(* IEC 61131-3 sources: repolevel_ST_code_completion/ground_truth/repoeval_can/readful_result, 4 files *)

(* ---- CAN_Send_Data_SWMC.st ---- *)
It seems like you've pasted a portion of the code multiple times, and it is incomplete in some places. However, I can help you analyze and understand the structure of the `CAN_Send_Data_SWMC` function based on the provided fragments.

### Overview of the `CAN_Send_Data_SWMC` Function

The `CAN_Send_Data_SWMC` function is designed to send CAN (Controller Area Network) messages based on the `SWMC_ID` input. It uses a `CASE` statement to determine which CAN channel (`C1`, `C2`, `C3`, etc.) to use for transmitting the message. The function takes the following inputs:
- `SWMC_ID`: A `UINT` value that determines which CAN channel to use.
- `id`: A `UINT` value used to calculate the `TxMsg_CobId`.
- `data`: An array of 8 bytes representing the data to be transmitted.

### Key Observations
1. **Message Structure**:
   - Each CAN channel (e.g., `C1TxMsg`, `C2TxMsg`, etc.) has a `TxMsg_CobId` and `TxMsg_Byte` field.
   - The `TxMsg_CobId` is calculated as `8 + 32 * id`.
   - The `TxMsg_Byte` is assigned the `data` array.

2. **Message Count and Counter**:
   - The `NoOfTxMessages` is set to `1` for each channel, indicating that one message is being transmitted.
   - The `TxCounter` is incremented by 1 for each transmission, likely to keep track of the number of messages sent.

3. **SWMC_ID Handling**:
   - The `CASE` statement handles different `SWMC_ID` values (e.g., `1`, `2`, `3`, `4`).
   - For each `SWMC_ID`, the corresponding CAN channel is selected, and the message is prepared for transmission.

### Issues in the Provided Code
1. **Incomplete Code**:
   - The code fragments are incomplete, with some parts cut off (e.g., the last fragment ends abruptly with `gCan.C1`).

2. **Redundancy**:
   - The same logic is repeated for each `SWMC_ID`. This could be refactored to reduce redundancy and improve maintainability.

3. **Missing Return Value**:
   - The function is declared to return a `BOOL`, but the return value is not shown in the provided code. It is unclear what the function should return (e.g., success/failure of the transmission).

### Refactored Version
Here’s a refactored version of the function to reduce redundancy:

```st
FUNCTION CAN_Send_Data_SWMC : BOOL
VAR_INPUT
	SWMC_ID : UINT;
	id 		: UINT;
	data	: ARRAY[1..8] OF BYTE;
END_VAR
VAR
	txMsgPointer : POINTER TO gCan.C1TxMsg; // Generic pointer to CAN message structure
END_VAR

CASE SWMC_ID OF
	1: txMsgPointer := ADR(gCan.C1TxMsg);
	2: txMsgPointer := ADR(gCan.C2TxMsg);
	3: txMsgPointer := ADR(gCan.C3TxMsg);
	4: txMsgPointer := ADR(gCan.C4TxMsg);
	ELSE
		RETURN FALSE; // Invalid SWMC_ID
END_CASE;

// Set message parameters
txMsgPointer^.TXMsg[1].TxMsg_CobId := 8 + 32 * id;
txMsgPointer^.TXMsg[1].TxMsg_Byte := data;
txMsgPointer^.NoOfTxMessages := 1;
txMsgPointer^.TxCounter := txMsgPointer^.TxCounter + 1;

RETURN TRUE; // Transmission setup successful
```

### Explanation of Refactored Code
1. **Generic Pointer**:
   - A pointer (`txMsgPointer`) is used to reference the appropriate CAN message structure (`C1TxMsg`, `C2TxMsg`, etc.) based on `SWMC_ID`.

2. **Error Handling**:
   - If an invalid `SWMC_ID` is provided, the function returns `FALSE`.

3. **Reduced Redundancy**:
   - The message preparation logic is written only once, reducing code duplication.

4. **Return Value**:
   - The function returns `TRUE` if the message setup is successful, or `FALSE` if an invalid `SWMC_ID` is provided.

Let me know if you need further clarification or assistance!

(* ---- CAN_Send_Data_SWMC_1.st ---- *)
It seems like you've pasted a portion of the code multiple times, and it is incomplete in some places. However, I can help you analyze and understand the structure of the `CAN_Send_Data_SWMC` function based on the provided fragments.

### Overview of the `CAN_Send_Data_SWMC` Function

The `CAN_Send_Data_SWMC` function is designed to send CAN (Controller Area Network) messages based on the `SWMC_ID` input. It uses a `CASE` statement to determine which CAN channel (`C1`, `C2`, `C3`, etc.) to use for transmitting the message. The function takes the following inputs:
- `SWMC_ID`: A `UINT` value that determines which CAN channel to use.
- `id`: A `UINT` value used to calculate the `TxMsg_CobId`.
- `data`: An array of 8 bytes representing the data to be transmitted.

### Key Observations
1. **Message Structure**:
   - Each CAN channel (e.g., `C1TxMsg`, `C2TxMsg`, etc.) has a `TxMsg_CobId` and `TxMsg_Byte` field.
   - The `TxMsg_CobId` is calculated as `8 + 32 * id`.
   - The `TxMsg_Byte` is assigned the `data` array.

2. **Message Count and Counter**:
   - The `NoOfTxMessages` is set to `1` for each channel, indicating that one message is being transmitted.
   - The `TxCounter` is incremented by 1 for each transmission, likely to keep track of the number of messages sent.

3. **SWMC_ID Handling**:
   - The `CASE` statement handles different `SWMC_ID` values (e.g., `1`, `2`, `3`, `4`).
   - For each `SWMC_ID`, the corresponding CAN channel is selected, and the message is prepared for transmission.

### Issues in the Provided Code
1. **Incomplete Code**:
   - The code fragments are incomplete, with some parts cut off (e.g., the last fragment ends abruptly with `gCan.C1`).

2. **Redundancy**:
   - The same logic is repeated for each `SWMC_ID`. This could be refactored to reduce redundancy and improve maintainability.

3. **Missing Return Value**:
   - The function is declared to return a `BOOL`, but the return value is not shown in the provided code. It is unclear what the function should return (e.g., success/failure of the transmission).

### Refactored Version
Here’s a refactored version of the function to reduce redundancy:

```st
FUNCTION CAN_Send_Data_SWMC : BOOL
VAR_INPUT
	SWMC_ID : UINT;
	id 		: UINT;
	data	: ARRAY[1..8] OF BYTE;
END_VAR
VAR
	txMsgPointer : POINTER TO gCan.C1TxMsg; // Generic pointer to CAN message structure
END_VAR

CASE SWMC_ID OF
	1: txMsgPointer := ADR(gCan.C1TxMsg);
	2: txMsgPointer := ADR(gCan.C2TxMsg);
	3: txMsgPointer := ADR(gCan.C3TxMsg);
	4: txMsgPointer := ADR(gCan.C4TxMsg);
	ELSE
		RETURN FALSE; // Invalid SWMC_ID
END_CASE;

// Set message parameters
txMsgPointer^.TXMsg[1].TxMsg_CobId := 8 + 32 * id;
txMsgPointer^.TXMsg[1].TxMsg_Byte := data;
txMsgPointer^.NoOfTxMessages := 1;
txMsgPointer^.TxCounter := txMsgPointer^.TxCounter + 1;

RETURN TRUE; // Transmission setup successful
```

### Explanation of Refactored Code
1. **Generic Pointer**:
   - A pointer (`txMsgPointer`) is used to reference the appropriate CAN message structure (`C1TxMsg`, `C2TxMsg`, etc.) based on `SWMC_ID`.

2. **Error Handling**:
   - If an invalid `SWMC_ID` is provided, the function returns `FALSE`.

3. **Reduced Redundancy**:
   - The message preparation logic is written only once, reducing code duplication.

4. **Return Value**:
   - The function returns `TRUE` if the message setup is successful, or `FALSE` if an invalid `SWMC_ID` is provided.

Let me know if you need further clarification or assistance!

(* ---- CAN_Read_Data_SWMC.st ---- *)
It seems you have provided a code fragment written in Structured Text (ST), a programming language commonly used in industrial automation and PLC programming. The code defines a function named `CAN_Read_Data_SWMC`, which processes CAN (Controller Area Network) messages based on the `SWMC_ID` input.

The function uses a `CASE` statement to handle different `SWMC_ID` values, each corresponding to a specific SWMC (presumably a subsystem or module). For each case, it extracts the `id` and `data` from the corresponding CAN message buffer (`gCan.CxRxMsg.RXMsg[I]`) and assigns them to the `frame` variable of type `Can_baseframe`.

### Key Observations:
1. **Input Variables**:
   - `SWMC_ID`: A `UINT` value representing the ID of the SWMC module to process.
   - `I`: A `UINT` value representing the index of the message in the receive buffer.

2. **Output**:
   - The function returns a `Can_baseframe` structure containing the `id` and `data` extracted from the CAN message.

3. **SWMC_ID Cases**:
   - Cases `1` to `6` handle specific SWMC modules (`SWMC-C1` to `SWMC-C6`).
   - For each case, the `id` is calculated as `(RxMsg_CobId - 8) / 32`, and the `data` is directly assigned from `RxMsg_Byte`.
   - The `ELSE` case handles any other `SWMC_ID` values by setting the `id` to `0` and clearing the `data` array.

4. **Commented-Out Code**:
   - Some parts of the code are commented out (e.g., the `//*` and `//(*)` comments). This might indicate incomplete or experimental code.

5. **Repetition**:
   - The code for each case is nearly identical, differing only in the source of the CAN message (`C1RxMsg`, `C2RxMsg`, etc.). This could potentially be refactored to reduce redundancy.

### Suggestions for Improvement:
1. **Refactoring**:
   - Use an array or mapping to store the `gCan.CxRxMsg` objects, allowing the `SWMC_ID` to directly index into the array. This would eliminate the need for repetitive `CASE` statements.

   Example:
   ```structured-text
   VAR
       RxMsgArray : ARRAY[1..6] OF Can_RxMsgType := [gCan.C1RxMsg, gCan.C2RxMsg, gCan.C3RxMsg, gCan.C4RxMsg, gCan.C5RxMsg, gCan.C6RxMsg];
   END_VAR

   IF SWMC_ID >= 1 AND SWMC_ID <= 6 THEN
       frame.id := (RxMsgArray[SWMC_ID].RXMsg[I].RxMsg_CobId - 8) / 32;
       frame.data := RxMsgArray[SWMC_ID].RXMsg[I].RxMsg_Byte;
   ELSE
       frame.id := 0;
       frame.data := [0, 0, 0, 0, 0, 0, 0, 0];
   END_IF
   ```

2. **Error Handling**:
   - Add error handling for invalid `SWMC_ID` values or out-of-bounds buffer indices (`I`).

3. **Documentation**:
   - Provide more detailed comments explaining the purpose of the function, the significance of the `id` calculation, and the structure of the `Can_baseframe` and `RxMsg` types.

4. **Testing**:
   - Ensure thorough testing of all cases, including edge cases (e.g., invalid `SWMC_ID` values, empty buffers).

If you have specific questions about the code or need further assistance, feel free to ask!

(* ---- CAN_Read_Data_SWMC_1.st ---- *)
It seems you have provided a code fragment written in Structured Text (ST), a programming language commonly used in industrial automation and PLC programming. The code defines a function named `CAN_Read_Data_SWMC`, which processes CAN (Controller Area Network) messages based on the `SWMC_ID` input.

The function uses a `CASE` statement to handle different `SWMC_ID` values, each corresponding to a specific SWMC (presumably a subsystem or module). For each case, it extracts the `id` and `data` from the corresponding CAN message buffer (`gCan.CxRxMsg.RXMsg[I]`) and assigns them to the `frame` variable of type `Can_baseframe`.

### Key Observations:
1. **Input Variables**:
   - `SWMC_ID`: A `UINT` value representing the ID of the SWMC module to process.
   - `I`: A `UINT` value representing the index of the message in the receive buffer.

2. **Output**:
   - The function returns a `Can_baseframe` structure containing the `id` and `data` extracted from the CAN message.

3. **SWMC_ID Cases**:
   - Cases `1` to `6` handle specific SWMC modules (`SWMC-C1` to `SWMC-C6`).
   - For each case, the `id` is calculated as `(RxMsg_CobId - 8) / 32`, and the `data` is directly assigned from `RxMsg_Byte`.
   - The `ELSE` case handles any other `SWMC_ID` values by setting the `id` to `0` and clearing the `data` array.

4. **Commented-Out Code**:
   - Some parts of the code are commented out (e.g., the `//*` and `//(*)` comments). This might indicate incomplete or experimental code.

5. **Repetition**:
   - The code for each case is nearly identical, differing only in the source of the CAN message (`C1RxMsg`, `C2RxMsg`, etc.). This could potentially be refactored to reduce redundancy.

### Suggestions for Improvement:
1. **Refactoring**:
   - Use an array or mapping to store the `gCan.CxRxMsg` objects, allowing the `SWMC_ID` to directly index into the array. This would eliminate the need for repetitive `CASE` statements.

   Example:
   ```structured-text
   VAR
       RxMsgArray : ARRAY[1..6] OF Can_RxMsgType := [gCan.C1RxMsg, gCan.C2RxMsg, gCan.C3RxMsg, gCan.C4RxMsg, gCan.C5RxMsg, gCan.C6RxMsg];
   END_VAR

   IF SWMC_ID >= 1 AND SWMC_ID <= 6 THEN
       frame.id := (RxMsgArray[SWMC_ID].RXMsg[I].RxMsg_CobId - 8) / 32;
       frame.data := RxMsgArray[SWMC_ID].RXMsg[I].RxMsg_Byte;
   ELSE
       frame.id := 0;
       frame.data := [0, 0, 0, 0, 0, 0, 0, 0];
   END_IF
   ```

2. **Error Handling**:
   - Add error handling for invalid `SWMC_ID` values or out-of-bounds buffer indices (`I`).

3. **Documentation**:
   - Provide more detailed comments explaining the purpose of the function, the significance of the `id` calculation, and the structure of the `Can_baseframe` and `RxMsg` types.

4. **Testing**:
   - Ensure thorough testing of all cases, including edge cases (e.g., invalid `SWMC_ID` values, empty buffers).

If you have specific questions about the code or need further assistance, feel free to ask!
